Omron Sysmac Studio project Prueba timer (Sysmac Studio 1.18.0.15, StandardProject)

# Controller new_Controller_0: NJ101-1020 version 1.13
Units and slaves: Alimentación : NJ-Px3001; CPU : NJ101-1020
Task PrimaryTask (priority 4, period or condition 2000): Programa0

VAR_GLOBAL
    Marcha : BOOL;  (* at ECAT://node#[100,1]/Input Bit 8 bits/Input Bit 00 *)
    Amarillo : BOOL;  (* at ECAT://node#[100,3]/Output Bit 8 bits/Output Bit 01 *)
    Verde : BOOL;  (* at ECAT://node#[100,3]/Output Bit 8 bits/Output Bit 02 *)
    Rojo : BOOL;  (* at ECAT://node#[100,3]/Output Bit 8 bits/Output Bit 03 *)
    x : INT := 5;  (* network input *)
    y : INT := 5;  (* network input *)
    enviar : BOOL;  (* network input *)
END_VAR

PROGRAM Programa0
VAR
    Aux1 : BOOL;
    Timer1 : TON;
    Aux2 : BOOL;
    T1 : TIME;
    Timer2 : TON;
    T2 : TIME;
    Aux3 : BOOL;
    Timer3 : TON;
    T3 : TIME;
    Aux4 : BOOL;
    Aux5 : BOOL;
    Timer4 : TON;
    T4 : TIME;
    Time1 : TIME;
    Time2 : TIME;
END_VAR
VAR_EXTERNAL
    Marcha : BOOL;
    Amarillo : BOOL;
    enviar : BOOL;
    x : INT;
    y : INT;
    Rojo : BOOL;
    Verde : BOOL;
END_VAR
VAR
    _p1 : BOOL;
END_VAR

(* Section Sección0: ladder, written here as Structured Text *)

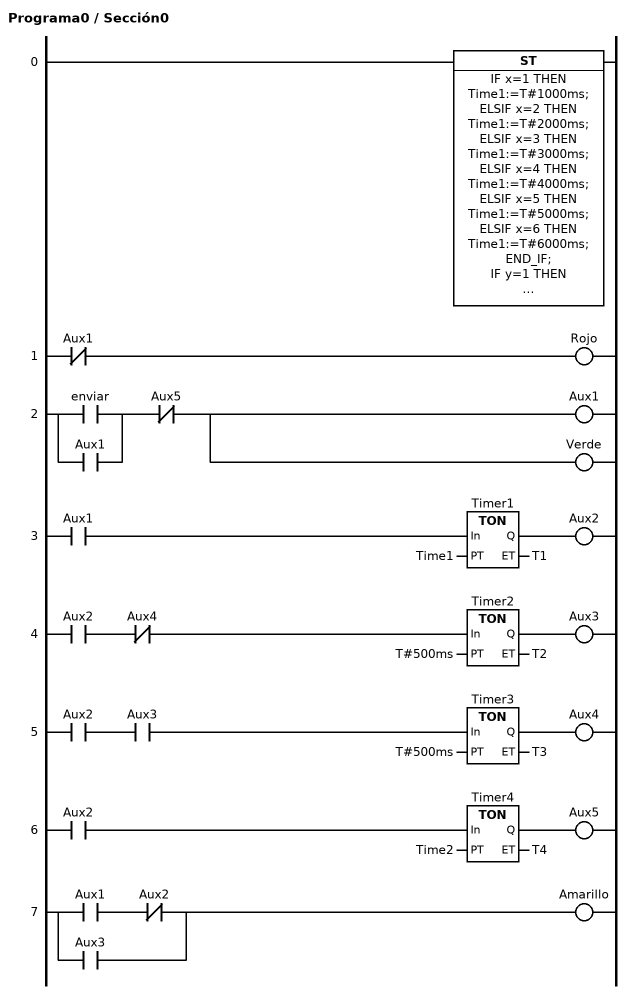
(* Rung 0 *)
IF x=1 THEN
	Time1:=T#1000ms;
ELSIF x=2 THEN
	Time1:=T#2000ms;
ELSIF x=3 THEN
	Time1:=T#3000ms;
ELSIF x=4 THEN
	Time1:=T#4000ms;
ELSIF x=5 THEN
	Time1:=T#5000ms;
ELSIF x=6 THEN
	Time1:=T#6000ms;
END_IF;


IF y=1 THEN
	Time2:=T#1000ms;
ELSIF y=2 THEN
	Time2:=T#2000ms;
ELSIF y=3 THEN
	Time2:=T#3000ms;
ELSIF y=4 THEN
	Time2:=T#4000ms;
ELSIF y=5 THEN
	Time2:=T#5000ms;
ELSIF y=6 THEN
	Time2:=T#6000ms;
END_IF;
(* Rung 1 *)
Rojo := NOT Aux1;
(* Rung 2 *)
_p1 := (enviar OR Aux1) AND NOT Aux5;
Aux1 := _p1;
Verde := _p1;
(* Rung 3 *)
Timer1(In := Aux1, PT := Time1, ET => T1);
Aux2 := Timer1.Q;
(* Rung 4 *)
Timer2(In := Aux2 AND NOT Aux4, PT := T#500ms, ET => T2);
Aux3 := Timer2.Q;
(* Rung 5 *)
Timer3(In := Aux2 AND Aux3, PT := T#500ms, ET => T3);
Aux4 := Timer3.Q;
(* Rung 6 *)
Timer4(In := Aux2, PT := Time2, ET => T4);
Aux5 := Timer4.Q;
(* Rung 7 *)
Amarillo := (Aux1 AND NOT Aux2) OR Aux3;
END_PROGRAM